(*********************************** G.D S.p.A. - Technical Department ***********************************
============= PROGRAM INFO ============
FOLDER:             TBD
MACHINES INVOLVED:  TBD 

============= DESCRIPTION =============

============= REVISIONS ===============
Date		Version	 	Author      	Description             
----------	-------		------------  	--------------------------------------------
2019/04/24 	0000.00	 	M.Grasso			Creation of the PRG

**********************************************************************************************************)
(*$R
	process_ref := prc;
$*)
PROGRAM csp_main_drives
VAR
	prc:						process;
	prc_path:					STRING;
	
		
END_VAR

VAR CONSTANT
	INCOHERENCE_TIMEOUT_MS:		INT := 2000;
END_VAR

_read_var_input();

_object_manager();

IF NOT objects_running()
THEN
	RETURN;	
END_IF

_read_process_image();

_mode_manager();

CASE process_get_mode(prc) of
	MODE_ABSENT,
	MODE_INACTIVE:
		RETURN;
	MODE_TEST:
		_handle_process_test();
END_CASE

_set_runtime_properties();

(********************************* BODY *********************************)

(************************************************************************)

_handle_messages();

_write_output();

ACTION _handle_messages:
;
END_ACTION

ACTION _handle_process_test:
;
END_ACTION

ACTION _mode_manager:
IF process_mode_req_is_pending(prc)
THEN
    process_apply_mode_req_first_step(prc);
    CASE process_get_mode(prc) OF
        MODE_TO_ABSENT:
			;
        MODE_TO_INACTIVE:
			;
        MODE_TO_TEST:
			;
        MODE_TO_OPERATIONAL:
			;
    END_CASE
    process_apply_mode_req_second_step(prc);
END_IF
END_ACTION

ACTION _object_manager:
IF objects_initialization()
THEN
	sub_process_init(
		object_name					:= 'csp_main_drives.prc', 
		process						:= csp_main.prc, 
		CONVERSION_this				:= prc);
		
	prc_path 						:= process_get_path(prc);

END_IF

IF objects_running()
THEN
	process_cycle(prc);
	
	
END_IF
END_ACTION

ACTION _read_process_image:
;
END_ACTION

ACTION _read_var_input:
;
END_ACTION

ACTION _set_runtime_properties:
;
END_ACTION

ACTION _write_output:
;
END_ACTION

END_PROGRAM

(* stored: Version 1.1.0.1, ProductVersion 3.1.4024.3
   POU csp_main_drives: Id {d167f5b5-c49e-408a-8a75-6d4be7374db4}, SpecialFunc None
   Action _handle_messages: Id {2ff567d2-4976-4429-995e-31007e7b7932}
   Action _handle_process_test: Id {974f7143-1730-405c-90d0-77110dd92a77}
   Action _mode_manager: Id {26846e1a-203a-488c-b556-ec4a42e03550}
   Action _object_manager: Id {afb92555-f0a9-4816-9867-4355dcb0f9eb}
   Action _read_process_image: Id {3b5815da-cfee-488e-8684-679c602d90aa}
   Action _read_var_input: Id {fc123db1-bdf2-4bd5-8b8e-f25a4f2410c9}
   Action _set_runtime_properties: Id {655226c7-1117-48ac-a5d5-7d88a512bc51}
   Action _write_output: Id {fa6c80bf-28d4-4162-8cc9-d7b96144124c} *)
